TYPE ST_AteqResultsRaw : //will be disregarded
STRUCT
    nProgramNumber              : WORD;     // Word 1
    nTestType                   : WORD;     // Word 2
    nRelayStatus                : WORD;     // Word 3 (bitmap)
    nAlarmCode                  : WORD;     // Word 4

    nPressureLowWord            : WORD;     // Word 5
    nPressureHighWord           : WORD;     // Word 6
    nPressureUnitCodeLowWord    : WORD;     // Word 7
    nPressureUnitCodeHighWord   : WORD;     // Word 8

    nLeakLowWord				: WORD;     // Word 9
    nLeakHighWord				: WORD;     // Word 10
    nLeakUnitCodeLowWord        : WORD;     // Word 11
    nLeakUnitCodeHighWord       : WORD;     // Word 12

    nPressurePiezo2LowWord              : WORD;     // Word 13
    nPressurePiezo2HighWord             : WORD;     // Word 14
    nPressurePiezo2UnitCodeLowWord      : WORD;     // Word 15
    nPressurePiezo2UnitCodeHighWord     : WORD;     // Word 16

    nTestCheckResultLowWord				: WORD;     // Word 17
    nTestCheckResultHighWord			: WORD;     // Word 18
    nTestCheckResultUnitCodeLowWord		: WORD;     // Word 19
    nTestCheckResultUnitCodeHighWord	: WORD;     // Word 20

    nLargeLeakLowWord           : WORD;     // Word 21
    nLargeLeakHighWord          : WORD;     // Word 22
    nLargeLeakUnitCodeLowWord   : WORD;     // Word 23
    nLargeLeakUnitCodeHighWord  : WORD;     // Word 24

    nPaLeakResultLowWord		: WORD;     // Word 25
    nPaLeakResultHighWord		: WORD;     // Word 26

    aReserved					: ARRAY[27..36] OF WORD; // Word 27-36 Unused

    nAtmPressureLowWord			: WORD;     // Word 37
    nAtmPressureHighWord		: WORD;     // Word 38
    nTempCelciusLowWord         : WORD;     // Word 39
    nTempCelciusHighWord        : WORD;     // Word 40

   	dtTestTimeStamp             : DT;       // Local time of reception
END_STRUCT
END_TYPE

(* stored: Version 1.1.0.1
   DUT ST_AteqResultsRaw: Id {3da4913a-8629-4ea8-bd6b-58104d8307fa} *)
